{attribute 'qualified_only'}
VAR_GLOBAL
    Axes :  ARRAY[1..4] OF AXIS_REF;
END_VAR

(* stored: Version 1.1.0.1
   GVL GVL_Axes: Id {b26e4e39-7a8c-452f-bac4-bbe855cef5f7} *)
